FUNCTION_BLOCK GateHandler EXTENDS BaseState
VAR_INPUT
END_VAR
VAR_OUTPUT
END_VAR
VAR
	InternalGateTime : TIME;
	InternalGateNumber : INT;
END_VAR

METHOD mIrun : BOOL
BasePointer^.GateAccessI[InternalGateNumber].mAutoOn();
StateTimer(IN:= TRUE, PT:=InternalGateTime);
IF StateTimer.Q THEN
	BasePointer^.GateAccessI[InternalGateNumber].mAutoOff();
	mNextState();
	StateTimer(IN:= FALSE);
END_IF
END_METHOD

METHOD mStateInit : BOOL
VAR_INPUT
	GateTime : TIME;
	GateNumber : INT;
END_VAR
InternalGateTime := GateTime;
InternalGateNumber := GateNumber;
END_METHOD

END_FUNCTION_BLOCK

(* stored: Version 1.1.0.1, ProductVersion 3.1.4024.12
   POU GateHandler: Id {fbb228c9-2aa9-4589-8773-a25047d3db88}, SpecialFunc None
   Method mIrun: Id {11921aaf-0c7e-4205-b4ae-86b3c762fae2}
   Method mStateInit: Id {3089b3ed-5b88-4954-9671-d016071c80bf} *)
